PROGRAM Cell_Main
VAR_INPUT
	
END_VAR

VAR_OUTPUT

END_VAR

Cell.StateManager();
Cell_Sequencer();
Comp01_Main();

END_PROGRAM

(* stored: Version 1.1.0.1, ProductVersion 3.1.4022.11
   POU Cell_Main: Id {44b70484-de62-433a-a258-7c9cb06da051}, SpecialFunc None *)
